			// Refresh active signal
			IF NOT _ServiceStates[nIndex].Alarm.Active THEN
				_ServiceStates[nIndex].Alarm.Active := TRUE;
				_ServiceStates[nIndex].Alarm.Acknowledged := FALSE;
				_ServiceStates[nIndex].Alarm.OccurrenceCount := _ServiceStates[nIndex].Alarm.OccurrenceCount + 1;
			END_IF
			M_ObserveServiceAlarm := TRUE;
			RETURN;
		END_IF

	// Update first empty slot index
	ELSIF nFirstEmpty = 0 THEN
		nFirstEmpty := nIndex;
	END_IF
END_FOR

IF nFirstEmpty = 0 THEN
	Overflow := TRUE;
	RETURN;
END_IF

M_LatchState(
	State := _ServiceStates[nFirstEmpty],
	Snapshot := Alarm,
	ServiceId := Alarm.ServiceId,
	DateTime := Alarm.DateTime);
_ServiceStates[nFirstEmpty].SeenThisCycle := TRUE;
M_ObserveServiceAlarm := TRUE;
END_METHOD

METHOD PUBLIC M_ProcessAcknowledgement
VAR_IN_OUT CONSTANT
	Request : ST_AlarmAckRequest;
END_VAR
VAR
	nIndex : UINT;
	bFound : BOOL;
END_VAR
_AckRequestOneShot(CLK := Request.bChangeRequest);

// Keep the response visible until the upper controller releases the request.
IF NOT Request.bChangeRequest THEN
	AckAccepted := FALSE;
	AckError := E_AlarmAckError.None;
	RETURN;
END_IF

IF NOT _AckRequestOneShot.Q THEN
	RETURN;
END_IF

AckResponseId := Request.RequestId;
AckAccepted := FALSE;
AckError := E_AlarmAckError.None;
bFound := FALSE;

IF Request.RequestId = 0 THEN
	AckError := E_AlarmAckError.InvalidRequestId;
	RETURN;
END_IF
IF Request.RequestId = _LastAckRequestId THEN
	AckError := E_AlarmAckError.DuplicateRequest;
	RETURN;
END_IF
_LastAckRequestId := Request.RequestId;

CASE Request.Command OF
	E_AlarmAckCommand.AcknowledgeOne:
		IF Request.MainErrorId = 0 THEN
			AckError := E_AlarmAckError.AlarmNotFound;
			RETURN;
		END_IF

		IF Request.ServiceId = 0 THEN
			FOR nIndex := 1 TO Param_Config.MaxConfiguredAlarmsPerModule DO
				IF _ConfiguredStates[nIndex].Latched
					AND (_ConfiguredStates[nIndex].Alarm.MainErrorId = Request.MainErrorId) THEN
					M_AcknowledgeState(State := _ConfiguredStates[nIndex]);
					bFound := TRUE;
					EXIT;
				END_IF
			END_FOR

			IF NOT bFound THEN
				FOR nIndex := 1 TO Param_Config.MaxHookAlarmsPerModule DO
					IF _HookStates[nIndex].Latched
						AND (_HookStates[nIndex].Alarm.MainErrorId = Request.MainErrorId) THEN
						M_AcknowledgeState(State := _HookStates[nIndex]);
						bFound := TRUE;
						EXIT;
					END_IF
				END_FOR
			END_IF
		ELSE
			FOR nIndex := 1 TO Param_Config.MaxServiceAlarmsPerModule DO
				IF _ServiceStates[nIndex].Latched
					AND (_ServiceStates[nIndex].Alarm.ServiceId = Request.ServiceId)
					AND (_ServiceStates[nIndex].Alarm.MainErrorId = Request.MainErrorId) THEN
					M_AcknowledgeState(State := _ServiceStates[nIndex]);
					bFound := TRUE;
					EXIT;
				END_IF
			END_FOR
		END_IF

		IF NOT bFound THEN
			AckError := E_AlarmAckError.AlarmNotFound;
			RETURN;
		END_IF

	E_AlarmAckCommand.AcknowledgeAll:
		FOR nIndex := 1 TO Param_Config.MaxConfiguredAlarmsPerModule DO
			IF _ConfiguredStates[nIndex].Latched THEN
				M_AcknowledgeState(State := _ConfiguredStates[nIndex]);
			END_IF
		END_FOR
		FOR nIndex := 1 TO Param_Config.MaxServiceAlarmsPerModule DO
			IF _ServiceStates[nIndex].Latched THEN
				M_AcknowledgeState(State := _ServiceStates[nIndex]);
			END_IF
		END_FOR

		FOR nIndex := 1 TO Param_Config.MaxHookAlarmsPerModule DO
			IF _HookStates[nIndex].Latched THEN
				M_AcknowledgeState(State := _HookStates[nIndex]);
			END_IF
		END_FOR
ELSE
	AckError := E_AlarmAckError.InvalidCommand;
	RETURN;
END_CASE

AckAccepted := TRUE;
END_METHOD

METHOD PUBLIC M_Publish
VAR_IN_OUT
	AlarmList : ARRAY[1..Param_Config.MaxPublishedModuleAlarms] OF ST_ExtAlarm;
END_VAR
VAR
	nIndex : UINT;
	nTarget : UINT;
END_VAR
MEMSET(ADR(AlarmList), 0, SIZEOF(AlarmList));
ConfiguredLatchedCount := 0;
ServiceLatchedCount := 0;
HookLatchedCount := 0;
nTarget := 1;

// Publish Service alarms first, configured alarms second, Hook alarms last.
FOR nIndex := 1 TO Param_Config.MaxServiceAlarmsPerModule DO
	IF NOT _ServiceStates[nIndex].Latched THEN
		CONTINUE;
	END_IF
	ServiceLatchedCount := ServiceLatchedCount + 1;
	IF nTarget > Param_Config.MaxPublishedModuleAlarms THEN
		Overflow := TRUE;
		CONTINUE;
	END_IF
	AlarmList[nTarget] := _ServiceStates[nIndex].Alarm;
	nTarget := nTarget + 1;
END_FOR

FOR nIndex := 1 TO Param_Config.MaxConfiguredAlarmsPerModule DO
	IF NOT _ConfiguredStates[nIndex].Latched THEN
		CONTINUE;
	END_IF
	ConfiguredLatchedCount := ConfiguredLatchedCount + 1;
	IF nTarget > Param_Config.MaxPublishedModuleAlarms THEN
		Overflow := TRUE;
		CONTINUE;
	END_IF
	AlarmList[nTarget] := _ConfiguredStates[nIndex].Alarm;
	nTarget := nTarget + 1;
END_FOR

FOR nIndex := 1 TO Param_Config.MaxHookAlarmsPerModule DO
	IF NOT _HookStates[nIndex].Latched THEN
		CONTINUE;
	END_IF
	HookLatchedCount := HookLatchedCount + 1;
	IF nTarget > Param_Config.MaxPublishedModuleAlarms THEN
		Overflow := TRUE;
		CONTINUE;
	END_IF
	AlarmList[nTarget] := _HookStates[nIndex].Alarm;
	nTarget := nTarget + 1;
END_FOR
END_METHOD

METHOD PRIVATE M_ResetAcknowledgement
AckResponseId := 0;
AckAccepted := FALSE;
AckError := E_AlarmAckError.None;
_LastAckRequestId := 0;
_AckRequestOneShot(CLK := FALSE);
END_METHOD

METHOD PUBLIC M_UpdateConfiguredAlarm
VAR_INPUT
	AlarmIndex : UINT;
	SampleValid : BOOL;
	ConditionMet : BOOL;
	UtcDateTime : STRING(20);
END_VAR
VAR_IN_OUT CONSTANT
	Alarm : ST_ExtAlarm;
END_VAR
IF (AlarmIndex < 1)
	OR (AlarmIndex > Param_Config.MaxConfiguredAlarmsPerModule)
	OR NOT SampleValid THEN
	RETURN;
END_IF

IF ConditionMet THEN
	IF NOT _ConfiguredStates[AlarmIndex].PreviousActive THEN
		IF NOT _ConfiguredStates[AlarmIndex].Latched THEN
			M_LatchState(
				State := _ConfiguredStates[AlarmIndex],
				Snapshot := Alarm,
				ServiceId := 0,
				DateTime := UtcDateTime);
		ELSE
			_ConfiguredStates[AlarmIndex].Alarm.Active := TRUE;
			_ConfiguredStates[AlarmIndex].Alarm.Acknowledged := FALSE;
			_ConfiguredStates[AlarmIndex].Alarm.OccurrenceCount := _ConfiguredStates[AlarmIndex].Alarm.OccurrenceCount + 1;
		END_IF
	END_IF
	_ConfiguredStates[AlarmIndex].Alarm.Active := TRUE;

ELSE
	IF _ConfiguredStates[AlarmIndex].PreviousActive
		AND _ConfiguredStates[AlarmIndex].Latched THEN
		_ConfiguredStates[AlarmIndex].Alarm.Active := FALSE;
		IF _ConfiguredStates[AlarmIndex].Alarm.Acknowledged THEN
			MEMSET(ADR(_ConfiguredStates[AlarmIndex]), 0, SIZEOF(_ConfiguredStates[AlarmIndex]));
		END_IF
	END_IF
END_IF

_ConfiguredStates[AlarmIndex].PreviousActive := ConditionMet;
END_METHOD

METHOD PUBLIC M_ObserveHookAlarm : BOOL
VAR_IN_OUT CONSTANT
	Alarm : ST_ExtAlarm;
END_VAR
VAR
	nIndex : UINT;
	nFirstEmpty : UINT;
END_VAR
M_ObserveHookAlarm := FALSE;
nFirstEmpty := 0;

IF (Alarm.ServiceId <> 0) OR (Alarm.MainErrorId = 0) THEN
	RETURN;
END_IF

FOR nIndex := 1 TO Param_Config.MaxHookAlarmsPerModule DO

	IF _HookStates[nIndex].Latched THEN

		IF (_HookStates[nIndex].Alarm.ServiceId = Alarm.ServiceId)
			AND (_HookStates[nIndex].Alarm.MainErrorId = Alarm.MainErrorId) THEN
			IF _HookStates[nIndex].SeenThisCycle THEN
				IF DuplicateId = 0 THEN
					DuplicateId := Alarm.MainErrorId;
				END_IF
				RETURN;
			END_IF
			_HookStates[nIndex].SeenThisCycle := TRUE;

			// A recurrence keeps the first snapshot and requires a fresh acknowledgement.
			IF NOT _HookStates[nIndex].Alarm.Active THEN
				_HookStates[nIndex].Alarm.Active := TRUE;
				_HookStates[nIndex].Alarm.Acknowledged := FALSE;
				_HookStates[nIndex].Alarm.OccurrenceCount := _HookStates[nIndex].Alarm.OccurrenceCount + 1;
			END_IF
			M_ObserveHookAlarm := TRUE;
			RETURN;
		END_IF

	// Reserve the first free slot without replacing a latched lifecycle.
	ELSIF nFirstEmpty = 0 THEN
		nFirstEmpty := nIndex;
	END_IF
END_FOR

IF nFirstEmpty = 0 THEN
	Overflow := TRUE;
	RETURN;
END_IF

M_LatchState(
	State := _HookStates[nFirstEmpty],
	Snapshot := Alarm,
	ServiceId := Alarm.ServiceId,
	DateTime := Alarm.DateTime);
_HookStates[nFirstEmpty].SeenThisCycle := TRUE;
M_ObserveHookAlarm := TRUE;
END_METHOD

METHOD PUBLIC M_SuppressHookAlarm
VAR_INPUT
	MainErrorId : UDINT;
END_VAR
VAR
	nIndex : UINT;
END_VAR
// Apply configuration ownership before acknowledgement, even when the source is invalid.
FOR nIndex := 1 TO Param_Config.MaxHookAlarmsPerModule DO
	IF _HookStates[nIndex].Latched AND (_HookStates[nIndex].Alarm.MainErrorId = MainErrorId) THEN
		MEMSET(ADR(_HookStates[nIndex]), 0, SIZEOF(_HookStates[nIndex]));
		RETURN;
	END_IF
END_FOR
END_METHOD

END_FUNCTION_BLOCK

// ---- POUs/10_Module/FB_ModuleBase.TcPOU
FUNCTION_BLOCK FB_ModuleBase EXTENDS FB_PackMLModeSet
VAR_INPUT
	ModuleCtrl : REFERENCE TO ST_ModuleCtrl;
	SystemContext : REFERENCE TO ST_SystemContext;
	HeartbeatIndex : UDINT;
	RuntimeConfig : REFERENCE TO ST_ModuleRuntimeConfig;
	VariableNodeReader : I_VariableNodeReader;
END_VAR

VAR_OUTPUT
	ModuleStatus : ST_ModuleStatus;
	ModuleVariableList : ARRAY[1..Param_Config.MaxModuleVariable] OF ST_ExtDescriptor;
	ModuleAlarmList : ARRAY[1..Param_Config.MaxPublishedModuleAlarms] OF ST_ExtAlarm;
	ModuleDataList : ARRAY[1..Param_Config.MaxModuleData] OF ST_ExtDescriptor;
END_VAR

VAR
	_CmdRequestOneShot : R_TRIG;
	_ModeRequestOneShot : R_TRIG;
	
	_ModuleId : UDINT;
	_ServiceContext : ST_ServiceContext;
	
	_HeartbeatTimer : TON;
	_LastHeartbeatIndex : UDINT;
	_IsControlSourceAlive : BOOL;
	_ConfiguredSnapshot : FB_ConfigValueSnapshotReader;
	_AlarmManager : FB_ModuleAlarmManager;
	_InAlarmHook : BOOL;
	_InVariableHook : BOOL;
	_ConfiguredVariableCount : UINT;
	_ServiceCoordinator : FB_ServiceCoordinator;
	_ServiceRegistrationAttempted : BOOL;
END_VAR

METHOD PROTECTED FINAL H_OnAborting : E_PackMLHookResult
VAR_INPUT
	bFirstScan : BOOL;
END_VAR
H_OnAborting := E_PackMLHookResult.Busy;
IF _ServiceCoordinator.AllAborted THEN
	H_OnAborting := E_PackMLHookResult.Done;
END_IF
END_METHOD

METHOD PROTECTED FINAL H_OnClearing : E_PackMLHookResult
VAR_INPUT
	bFirstScan : BOOL;
END_VAR
H_OnClearing := E_PackMLHookResult.Busy;
IF _ServiceCoordinator.AllStopped THEN
	H_OnClearing := E_PackMLHookResult.Done;
END_IF
END_METHOD

METHOD PROTECTED FINAL H_OnIdle
VAR_INPUT
	bFirstScan	: BOOL;
END_VAR
// Transfer to execute automatically
RequestCommand(E_PackMLCommand.Start);
END_METHOD

METHOD PROTECTED FINAL H_OnResetting : E_PackMLHookResult
VAR_INPUT
	bFirstScan : BOOL;
END_VAR
H_OnResetting := E_PackMLHookResult.Busy;
IF _ServiceCoordinator.AllIdle THEN
	H_OnResetting := E_PackMLHookResult.Done;
END_IF
END_METHOD

METHOD PROTECTED FINAL H_OnStopping : E_PackMLHookResult
VAR_INPUT
	bFirstScan : BOOL;
END_VAR
H_OnStopping := E_PackMLHookResult.Busy;
IF _ServiceCoordinator.AllStopped THEN
	H_OnStopping := E_PackMLHookResult.Done;
END_IF
END_METHOD

METHOD PROTECTED H_RegisterServices
// Derived Modules register persistent Service storage once.
END_METHOD

METHOD PROTECTED H_UpdateAlarm
// Optional Module extension; submitted values belong to this scan.
END_METHOD

METHOD PROTECTED H_UpdateBaseUnit
VAR_INPUT
END_VAR
END_METHOD

METHOD PROTECTED H_UpdateService
VAR_INPUT
END_VAR
END_METHOD

METHOD PROTECTED H_UpdateVariable
// Optional Module extension; submitted values belong to this scan.
END_METHOD

METHOD PROTECTED FINAL M_AddAlarm : BOOL
VAR_INPUT
	MainErrorId : UDINT;
	SourceErrorId : UDINT;
	Message : STRING;
	Path : STRING(255);
	Severity : E_Severity;
END_VAR
VAR
	nIndex : UINT;
	Alarm : ST_ExtAlarm;
END_VAR
M_AddAlarm := FALSE;
IF NOT _InAlarmHook OR (MainErrorId = 0) THEN
	RETURN;
END_IF
IF __ISVALIDREF(RuntimeConfig) THEN
	IF RuntimeConfig.Valid THEN
		FOR nIndex := 1 TO RuntimeConfig.AlarmCount DO
			IF RuntimeConfig.AlarmBindings[nIndex].Definition.MainErrorId = MainErrorId THEN
				M_AddAlarm := TRUE; // JSON owns the complete definition, even without a valid sample.
				RETURN;
			END_IF
		END_FOR
	END_IF
END_IF
MEMSET(ADR(Alarm), 0, SIZEOF(Alarm));
Alarm.MainErrorId := MainErrorId;
Alarm.SourceErrorId := SourceErrorId;
Alarm.Message := Message;
Alarm.Path := Path;
Alarm.Severity := Severity;
Alarm.DateTime := _ServiceContext.UtcDateTime;
M_AddAlarm := _AlarmManager.M_ObserveHookAlarm(Alarm := Alarm);
END_METHOD

METHOD PROTECTED FINAL M_AddVariable : BOOL
VAR_INPUT
	Id : UDINT;
	Name : STRING(30);
	DataType : E_DescriptorType;
	Unit : STRING(10);
	Value : STRING(80);
END_VAR
VAR
	nIndex : UINT;
END_VAR
M_AddVariable := FALSE;
IF NOT _InVariableHook OR (Id = 0) THEN
	RETURN;
END_IF
FOR nIndex := 1 TO ModuleStatus.Variable.PublishedCount DO
	IF ModuleVariableList[nIndex].Id = Id THEN
		IF nIndex <= _ConfiguredVariableCount THEN
			M_AddVariable := TRUE; // JSON ownership is not a duplicate submission.
		ELSIF ModuleStatus.Variable.DuplicateId = 0 THEN
			ModuleStatus.Variable.DuplicateId := Id;
		END_IF
		RETURN;
	END_IF
END_FOR
IF ModuleStatus.Variable.PublishedCount >= Param_Config.MaxModuleVariable THEN
	ModuleStatus.Variable.Overflow := TRUE;
	RETURN;
END_IF
ModuleStatus.Variable.PublishedCount := ModuleStatus.Variable.PublishedCount + 1;
nIndex := ModuleStatus.Variable.PublishedCount;
ModuleVariableList[nIndex].Id := Id;
ModuleVariableList[nIndex].Name := Name;
ModuleVariableList[nIndex].DataType := DataType;
ModuleVariableList[nIndex].Unit := Unit;
ModuleVariableList[nIndex].Value := Value;
M_AddVariable := TRUE;
END_METHOD

METHOD PRIVATE M_CheckHeartbeat
VAR_INPUT
END_VAR

VAR
	bLooseHeartbeat : BOOL;
	HeartbeatTimeout : TIME;
END_VAR
HeartbeatTimeout := SystemContext.ModuleHeartbeatTimeout;
IF HeartbeatTimeout <= T#0S THEN
	HeartbeatTimeout := Param_Config.ModuleHeartbeat_Timeout;
END_IF

// Heartbeats check
bLooseHeartbeat := _LastHeartbeatIndex = HeartbeatIndex;
IF bLooseHeartbeat THEN
	_HeartbeatTimer(IN := TRUE, PT := HeartbeatTimeout);
ELSE
	_HeartbeatTimer(IN := FALSE, PT := HeartbeatTimeout);
END_IF

// Update Last Heartbeat Index
_LastHeartbeatIndex := HeartbeatIndex;

// Update Is ControlSource Alive status
_IsControlSourceAlive := NOT _HeartbeatTimer.Q;
END_METHOD

METHOD PRIVATE M_PublishAlarmState
_AlarmManager.M_Publish(AlarmList := ModuleAlarmList);
ModuleStatus.Alarm.AckResponseId := _AlarmManager.AckResponseId;
ModuleStatus.Alarm.AckAccepted := _AlarmManager.AckAccepted;
ModuleStatus.Alarm.AckError := _AlarmManager.AckError;
ModuleStatus.Alarm.ConfiguredLatchedCount := _AlarmManager.ConfiguredLatchedCount;
ModuleStatus.Alarm.Overflow := _AlarmManager.Overflow;
ModuleStatus.Alarm.ServiceLatchedCount := _AlarmManager.ServiceLatchedCount;
ModuleStatus.Alarm.HookLatchedCount := _AlarmManager.HookLatchedCount;
ModuleStatus.Alarm.DuplicateId := _AlarmManager.DuplicateId;
END_METHOD

METHOD PROTECTED FINAL M_RegisterService : BOOL
VAR_INPUT
	ServiceId : UDINT;
	AllowCompositeCall : BOOL;
	UpperParam : ANY;
	EffectiveParam : ANY;
END_VAR
VAR_IN_OUT
	UpperCtrl : ST_ServiceCtrl;
	EffectiveCtrl : ST_ServiceCtrl;
	Status : ST_ServiceStatus;
END_VAR
M_RegisterService := _ServiceCoordinator.M_Register(
	ServiceId := ServiceId,
	AllowCompositeCall := AllowCompositeCall,
	UpperCtrl := UpperCtrl,
	EffectiveCtrl := EffectiveCtrl,
	UpperParam := UpperParam,
	EffectiveParam := EffectiveParam,
	Status := Status);
END_METHOD

METHOD PRIVATE M_UpdateAlarmState
VAR
	nAlarm : UINT;
	nSource : UINT;
	nRevision : UDINT;
	fValue : LREAL;
	bValid : BOOL;
	bConditionMet : BOOL;
	Alarm : ST_ExtAlarm;
END_VAR
nRevision := 0;
IF __ISVALIDREF(RuntimeConfig) THEN
	IF RuntimeConfig.Valid THEN
		nRevision := RuntimeConfig.Revision;
	END_IF
END_IF
_AlarmManager.M_BeginCycle(
	ModuleId := _ModuleId,
	ConfigurationRevision := nRevision);

// Remove identities now owned by JSON before an acknowledgement can find a stale Hook event.
IF __ISVALIDREF(RuntimeConfig) THEN
	IF RuntimeConfig.Valid THEN
		FOR nAlarm := 1 TO RuntimeConfig.AlarmCount DO
			_AlarmManager.M_SuppressHookAlarm(
				MainErrorId := RuntimeConfig.AlarmBindings[nAlarm].Definition.MainErrorId);
		END_FOR
	END_IF
END_IF

// Process acknowledgements before evaluating this cycle so AckAll cannot consume
// a new event that the upper controller has not observed yet.
_AlarmManager.M_ProcessAcknowledgement(Request := ModuleCtrl.AlarmAckRequest);

IF __ISVALIDREF(RuntimeConfig) THEN
	IF RuntimeConfig.Valid AND _ConfiguredSnapshot.Ready THEN
		FOR nAlarm := 1 TO RuntimeConfig.AlarmCount DO
			nSource := RuntimeConfig.VariableCount + nAlarm;
			fValue := _ConfiguredSnapshot.M_GetLReal(SourceIndex := nSource, Valid => bValid);
			bConditionMet := FALSE;
			IF bValid THEN
				bConditionMet := F_AlarmConditionMet(
					Value := fValue,
					Operator := RuntimeConfig.AlarmBindings[nAlarm].Definition.Operator,
					Threshold := RuntimeConfig.AlarmBindings[nAlarm].Definition.Threshold,
					Tolerance := RuntimeConfig.AlarmBindings[nAlarm].Definition.Tolerance);
			END_IF

			MEMSET(ADR(Alarm), 0, SIZEOF(Alarm));
			Alarm.ModuleId := _ModuleId;
			Alarm.ServiceId := 0;
			Alarm.MainErrorId := RuntimeConfig.AlarmBindings[nAlarm].Definition.MainErrorId;
			Alarm.SourceErrorId := RuntimeConfig.AlarmBindings[nAlarm].Definition.SourceErrorId;
			Alarm.Message := RuntimeConfig.AlarmBindings[nAlarm].Definition.Message;
			Alarm.Path := RuntimeConfig.AlarmBindings[nAlarm].Definition.Source;
			Alarm.Severity := RuntimeConfig.AlarmBindings[nAlarm].Definition.Severity;
			_AlarmManager.M_UpdateConfiguredAlarm(
				AlarmIndex := nAlarm,
				SampleValid := bValid,
				ConditionMet := bConditionMet,
				Alarm := Alarm,
				UtcDateTime := _ServiceContext.UtcDateTime);
		END_FOR
	END_IF
END_IF

_InAlarmHook := TRUE;
H_UpdateAlarm();
_InAlarmHook := FALSE;

M_UpdateServiceAlarms();
_AlarmManager.M_EndCycle();
END_METHOD

METHOD PRIVATE M_UpdateConfiguredVariableList
VAR
	nVariable : UINT;
	bValid : BOOL;
END_VAR
IF NOT __ISVALIDREF(RuntimeConfig) THEN
	RETURN;
END_IF
IF NOT RuntimeConfig.Valid THEN
	RETURN;
END_IF

FOR nVariable := 1 TO RuntimeConfig.VariableCount DO
	ModuleVariableList[nVariable].Id := RuntimeConfig.VariableBindings[nVariable].Definition.Id;
	ModuleVariableList[nVariable].Name := RuntimeConfig.VariableBindings[nVariable].Definition.Name;
	ModuleVariableList[nVariable].DataType := F_ConfigDataTypeToDescriptor(
		DataType := RuntimeConfig.VariableBindings[nVariable].Definition.DataType);
	ModuleVariableList[nVariable].Unit := RuntimeConfig.VariableBindings[nVariable].Definition.Unit;
	ModuleVariableList[nVariable].Value := _ConfiguredSnapshot.M_GetValueString(
		SourceIndex := nVariable,
		Valid => bValid);
END_FOR
_ConfiguredVariableCount := RuntimeConfig.VariableCount;
ModuleStatus.Variable.PublishedCount := _ConfiguredVariableCount;
END_METHOD

METHOD PROTECTED FINAL M_UpdateModule
IF NOT _ServiceRegistrationAttempted THEN
	_ServiceRegistrationAttempted := TRUE;
	_ServiceCoordinator.M_BeginRegistration();
	H_RegisterServices();
	_ServiceCoordinator.M_Seal();
END_IF

M_CheckHeartbeat();
ModuleStatus.IsControlSourceAlive := _IsControlSourceAlive;

// Update module state machine
PackMLIn := ModuleCtrl.PackMLIn;
SUPER^();

IF __ISVALIDREF(RuntimeConfig) THEN
	_ModuleId := RuntimeConfig.ModuleId;
	_ConfiguredSnapshot(
		RuntimeConfig := RuntimeConfig,
		VariableNodeReader := VariableNodeReader);
	ModuleStatus.ModuleId := _ModuleId;
	ModuleStatus.Enabled := RuntimeConfig.Enabled;
	ModuleStatus.ModuleType := RuntimeConfig.ModuleType;
END_IF

_ServiceContext.ModuleId := _ModuleId;
_ServiceContext.UtcDateTime := SystemContext.UtcDateTime;

// Update service state machine
_ServiceCoordinator.M_PrepareCycle(
	ModuleInExecute := PackMLOut.eStateCurrent = E_PackMLState.Execute,
	ModuleCtrl := ModuleCtrl);
H_UpdateService();

// Update base unit state machine
H_UpdateBaseUnit();

// Capture the status set produced by this scan for framework aggregation and
// for the Module PackML transition checks in the next scan.
_ServiceCoordinator.M_ObserveCycle();

_CmdRequestOneShot(CLK:= PackMLIn.bCommandChangeRequest, Q=> );
_ModeRequestOneShot(CLK:= PackMLIn.bModeChangeRequest, Q=> );

// Updata status
IF _CmdRequestOneShot.Q OR _ModeRequestOneShot.Q THEN
	ModuleStatus.ResponseId := ModuleCtrl.RequestId;
END_IF
ModuleStatus.PackMLOut := PackMLOut;

M_UpdateAlarmState();
M_PublishAlarmState();
M_UpdateServiceDataList();
M_UpdateVariableList();
END_METHOD

METHOD PRIVATE M_UpdateServiceAlarms
VAR
	nServiceIndex : UINT;
	nErrorIndex : UINT;
	ServiceStatus : ST_ServiceStatus;
END_VAR
// Submit currently observable Service errors. The manager owns lifecycle state
// and marks identities not observed in this scan inactive during M_EndCycle.
FOR nServiceIndex := 1 TO _ServiceCoordinator.RegisteredCount DO
	IF NOT _ServiceCoordinator.M_GetServiceStatusByIndex(
		Index := nServiceIndex,
		Status => ServiceStatus) THEN
		CONTINUE;
	END_IF
	FOR nErrorIndex := 1 TO Param_Config.MaxServiceError DO
		IF ServiceStatus.ErrorList[nErrorIndex].MainErrorId <> 0 THEN
			_AlarmManager.M_ObserveServiceAlarm(
				Alarm := ServiceStatus.ErrorList[nErrorIndex]);
		END_IF
	END_FOR
END_FOR
END_METHOD

METHOD PRIVATE M_UpdateServiceDataList
VAR
	nServiceIndex : UINT;
	nDataIndex : UINT;
	nPublishedIndex : UINT;
	bDuplicate : BOOL;
	DataId : UDINT;
	ServiceStatus : ST_ServiceStatus;
END_VAR
MEMSET(ADR(ModuleDataList), 0, SIZEOF(ModuleDataList));
MEMSET(ADR(ModuleStatus.Data), 0, SIZEOF(ModuleStatus.Data));

FOR nServiceIndex := 1 TO _ServiceCoordinator.RegisteredCount DO
	IF NOT _ServiceCoordinator.M_GetServiceStatusByIndex(
		Index := nServiceIndex,
		Status => ServiceStatus) THEN
		CONTINUE;
	END_IF
	IF ServiceStatus.Data.Overflow THEN
		ModuleStatus.Data.Overflow := TRUE;
	END_IF

	FOR nDataIndex := 1 TO Param_Config.MaxServiceData DO
		DataId := ServiceStatus.Data.DataList[nDataIndex].Id;
		IF DataId = 0 THEN
			CONTINUE;
		END_IF

		bDuplicate := FALSE;
		FOR nPublishedIndex := 1 TO ModuleStatus.Data.PublishedCount DO
			IF ModuleDataList[nPublishedIndex].Id = DataId THEN
				bDuplicate := TRUE;
				EXIT;
			END_IF
		END_FOR

		IF bDuplicate THEN
			IF ModuleStatus.Data.DuplicateId = 0 THEN
				ModuleStatus.Data.DuplicateId := DataId;
			END_IF
			CONTINUE;
		END_IF

		IF ModuleStatus.Data.PublishedCount >= Param_Config.MaxModuleData THEN
			ModuleStatus.Data.Overflow := TRUE;
			CONTINUE;
		END_IF

		ModuleStatus.Data.PublishedCount := ModuleStatus.Data.PublishedCount + 1;
		ModuleDataList[ModuleStatus.Data.PublishedCount] :=
			ServiceStatus.Data.DataList[nDataIndex];
	END_FOR
END_FOR
END_METHOD

METHOD PRIVATE M_UpdateVariableList
MEMSET(ADR(ModuleVariableList), 0, SIZEOF(ModuleVariableList));
MEMSET(ADR(ModuleStatus.Variable), 0, SIZEOF(ModuleStatus.Variable));
_ConfiguredVariableCount := 0;
M_UpdateConfiguredVariableList();
_InVariableHook := TRUE;
H_UpdateVariable();
_InVariableHook := FALSE;
END_METHOD

END_FUNCTION_BLOCK

// ---- POUs/10_Module/FB_ServiceCoordinator.TcPOU
FUNCTION_BLOCK FB_ServiceCoordinator
VAR
	_Entries : ARRAY[1..Param_Config.MaxServicesPerModule] OF ST_ServiceRegistrationEntry;
	_RegisteredCount : UINT;
	_RegistrationStarted : BOOL;
	_Sealed : BOOL;
	_RegistrationError : E_ServiceRegistrationError;
	_FailedServiceId : UDINT;
	_AllIdle : BOOL;
	_AllStopped : BOOL;
	_AllAborted : BOOL;
	_JsonDataType : FB_JsonReadWriteDataType;
END_VAR

PROPERTY PUBLIC FINAL AllAborted : BOOL
GET
AllAborted := _AllAborted;
END_GET
END_PROPERTY

PROPERTY PUBLIC FINAL AllIdle : BOOL
GET
AllIdle := _AllIdle;
END_GET
END_PROPERTY

PROPERTY PUBLIC FINAL AllStopped : BOOL
GET
AllStopped := _AllStopped;
END_GET
END_PROPERTY

PROPERTY PUBLIC FINAL FailedServiceId : UDINT
GET
FailedServiceId := _FailedServiceId;
END_GET
END_PROPERTY

METHOD PUBLIC FINAL M_BeginRegistration : BOOL
M_BeginRegistration := FALSE;
IF _RegistrationStarted THEN
	M_SetRegistrationError(Error := E_ServiceRegistrationError.RegistrationAlreadyStarted, ServiceId := 0);
	RETURN;
END_IF
MEMSET(ADR(_Entries), 0, SIZEOF(_Entries));
_RegisteredCount := 0;
_Sealed := FALSE;
_RegistrationError := E_ServiceRegistrationError.None;
_FailedServiceId := 0;
_AllIdle := FALSE;
_AllStopped := FALSE;
_AllAborted := FALSE;
_RegistrationStarted := TRUE;
M_BeginRegistration := TRUE;
END_METHOD

METHOD PRIVATE M_FindIndexByServiceId : UINT
VAR_INPUT
	ServiceId : UDINT;
END_VAR
VAR
	nIndex : UINT;
END_VAR
M_FindIndexByServiceId := 0;
IF ServiceId = 0 THEN RETURN; END_IF
FOR nIndex := 1 TO _RegisteredCount DO
	IF _Entries[nIndex].InUse AND (_Entries[nIndex].ServiceId = ServiceId) THEN
		M_FindIndexByServiceId := nIndex;
		RETURN;
	END_IF
END_FOR
END_METHOD

METHOD PUBLIC FINAL M_GetCompositeOwnershipState : E_CompositeOwnershipState
VAR_INPUT
	CompositeServiceId : UDINT;
END_VAR
VAR
	nIndex : UINT;
END_VAR
M_GetCompositeOwnershipState := E_CompositeOwnershipState.None;
nIndex := M_FindIndexByServiceId(ServiceId := CompositeServiceId);
IF (nIndex = 0) OR NOT _Entries[nIndex].IsComposite THEN RETURN; END_IF
M_GetCompositeOwnershipState := _Entries[nIndex].OwnershipState;
END_METHOD

METHOD PUBLIC FINAL M_GetInternalCommandState : E_ServiceInternalCommandState
VAR_INPUT
	CallerServiceId : UDINT;
	TargetServiceId : UDINT;
END_VAR
VAR
	nCallerIndex : UINT;
	nTargetIndex : UINT;
END_VAR
M_GetInternalCommandState := E_ServiceInternalCommandState.None;
nCallerIndex := M_FindIndexByServiceId(ServiceId := CallerServiceId);
nTargetIndex := M_FindIndexByServiceId(ServiceId := TargetServiceId);
IF (nCallerIndex = 0) OR (nTargetIndex = 0) THEN RETURN; END_IF
IF NOT M_IsDeclaredDependency(CompositeIndex := nCallerIndex, TargetServiceId := TargetServiceId) THEN RETURN; END_IF
IF (_Entries[nTargetIndex].CompositeOwnerServiceId <> CallerServiceId)
	AND (_Entries[nTargetIndex].InternalCommandState <> E_ServiceInternalCommandState.Cancelled) THEN RETURN; END_IF
M_GetInternalCommandState := _Entries[nTargetIndex].InternalCommandState;
END_METHOD

METHOD PUBLIC FINAL M_GetServiceSnapshotById : BOOL
VAR_INPUT
	ServiceId : UDINT;
END_VAR
VAR_OUTPUT
	Snapshot : ST_ServiceExecutionSnapshot;
END_VAR
VAR
	nIndex : UINT;
END_VAR
M_GetServiceSnapshotById := FALSE;
MEMSET(ADR(Snapshot), 0, SIZEOF(Snapshot));
nIndex := M_FindIndexByServiceId(ServiceId := ServiceId);
IF nIndex = 0 THEN RETURN; END_IF
Snapshot := _Entries[nIndex].ObservedSnapshot;
M_GetServiceSnapshotById := Snapshot.Valid;
END_METHOD

METHOD PUBLIC FINAL M_GetServiceStatusByIndex : BOOL
VAR_INPUT
	Index : UINT;
END_VAR
VAR_OUTPUT
	Status : ST_ServiceStatus;
END_VAR
VAR
	pStatus : POINTER TO ST_ServiceStatus;
END_VAR
M_GetServiceStatusByIndex := FALSE;
MEMSET(ADR(Status), 0, SIZEOF(Status));
IF (Index = 0) OR (Index > _RegisteredCount) THEN RETURN; END_IF
IF NOT _Entries[Index].InUse OR (_Entries[Index].StatusAddress = 0) THEN RETURN; END_IF
pStatus := _Entries[Index].StatusAddress;
Status := pStatus^;
M_GetServiceStatusByIndex := TRUE;
END_METHOD

METHOD PRIVATE M_IsDeclaredDependency : BOOL
VAR_INPUT
	CompositeIndex : UINT;
	TargetServiceId : UDINT;
END_VAR
VAR
	nDependency : UINT;
	pDependencies : POINTER TO UDINT;
END_VAR
M_IsDeclaredDependency := FALSE;
IF (CompositeIndex = 0) OR (CompositeIndex > _RegisteredCount)
	OR NOT _Entries[CompositeIndex].IsComposite
	OR (_Entries[CompositeIndex].CompositeDependenciesAddress = 0) THEN RETURN; END_IF

pDependencies := _Entries[CompositeIndex].CompositeDependenciesAddress;
FOR nDependency := 1 TO _Entries[CompositeIndex].CompositeDependencyCount DO
	IF pDependencies[nDependency - 1] = TargetServiceId THEN
		M_IsDeclaredDependency := TRUE;
		RETURN;
	END_IF
END_FOR
END_METHOD

METHOD PUBLIC FINAL M_ObserveCycle
VAR
	nIndex : UINT;
	pStatus : POINTER TO ST_ServiceStatus;
END_VAR
_AllIdle := FALSE;
_AllStopped := FALSE;
_AllAborted := FALSE;
IF NOT Ready OR (_RegisteredCount = 0) THEN RETURN; END_IF
_AllIdle := TRUE;
_AllStopped := TRUE;
_AllAborted := TRUE;
FOR nIndex := 1 TO _RegisteredCount DO
	pStatus := _Entries[nIndex].StatusAddress;
	_Entries[nIndex].ObservedSnapshot.Valid := TRUE;
	_Entries[nIndex].ObservedSnapshot.ServiceId := _Entries[nIndex].ServiceId;
	_Entries[nIndex].ObservedSnapshot.ResponseId := pStatus^.ResponseId;
	_Entries[nIndex].ObservedSnapshot.PackMLOut := pStatus^.PackMLOut;
	_Entries[nIndex].ObservedSnapshot.ExecuteSubState := pStatus^.ExecuteSubState;
	_Entries[nIndex].ObservedSnapshot.CompletionBehavior := pStatus^.CompletionBehavior;
	IF (_Entries[nIndex].InternalCommandState = E_ServiceInternalCommandState.RequestHigh)
		AND (pStatus^.ResponseId = _Entries[nIndex].InternalRequestId) THEN
		IF pStatus^.PackMLOut.bCommandAccepted THEN
			_Entries[nIndex].InternalCommandState := E_ServiceInternalCommandState.Accepted;
			_Entries[nIndex].InternalRequestMustGoLow := TRUE;
		ELSIF pStatus^.PackMLOut.bCommandRejected THEN
			_Entries[nIndex].InternalCommandState := E_ServiceInternalCommandState.Rejected;
			_Entries[nIndex].InternalRequestMustGoLow := TRUE;
		END_IF
	END_IF
	_AllIdle := _AllIdle AND (pStatus^.PackMLOut.eStateCurrent = E_PackMLState.Idle);
	_AllStopped := _AllStopped AND (pStatus^.PackMLOut.eStateCurrent = E_PackMLState.Stopped);
	_AllAborted := _AllAborted AND (pStatus^.PackMLOut.eStateCurrent = E_PackMLState.Aborted);
END_FOR
END_METHOD

METHOD PUBLIC FINAL M_PrepareCycle
VAR_INPUT
	ModuleInExecute : BOOL;
	ModuleCtrl : REFERENCE TO ST_ModuleCtrl;
END_VAR
VAR
	nIndex : UINT;
	pUpperCtrl : POINTER TO ST_ServiceCtrl;
	pEffectiveCtrl : POINTER TO ST_ServiceCtrl;
	bUpperCommandHigh : BOOL;
	bUpperModeHigh : BOOL;
	bNewStartRequest : BOOL;
END_VAR
IF Ready AND ModuleInExecute THEN
	M_ProcessOwnershipRequests();
ELSIF Ready THEN
	FOR nIndex := 1 TO _RegisteredCount DO
		IF _Entries[nIndex].OwnershipState = E_CompositeOwnershipState.Pending THEN
			_Entries[nIndex].OwnershipState := E_CompositeOwnershipState.Cancelled;
		END_IF
	END_FOR
END_IF
FOR nIndex := 1 TO _RegisteredCount DO
	pUpperCtrl := _Entries[nIndex].UpperCtrlAddress;
	pEffectiveCtrl := _Entries[nIndex].EffectiveCtrlAddress;
	IF NOT Ready THEN
		pEffectiveCtrl^.PackMLIn.bCommandChangeRequest := FALSE;
		pEffectiveCtrl^.PackMLIn.bModeChangeRequest := FALSE;
		CONTINUE;
	END_IF
	bUpperCommandHigh := pUpperCtrl^.PackMLIn.bCommandChangeRequest;
	bUpperModeHigh := pUpperCtrl^.PackMLIn.bModeChangeRequest;
	IF NOT ModuleInExecute THEN
		IF (_Entries[nIndex].InternalCommandState = E_ServiceInternalCommandState.Queued)
			OR (_Entries[nIndex].InternalCommandState = E_ServiceInternalCommandState.RequestHigh)
			OR _Entries[nIndex].InternalRequestMustGoLow THEN
			_Entries[nIndex].InternalCommandState := E_ServiceInternalCommandState.Cancelled;
			_Entries[nIndex].InternalRequestMustGoLow := FALSE;
		END_IF
		pEffectiveCtrl^.RequestId := ModuleCtrl.RequestId;
		pEffectiveCtrl^.PackMLIn := ModuleCtrl.PackMLIn;
		IF bUpperCommandHigh THEN _Entries[nIndex].UpperCommandBlockedUntilFalse := TRUE; END_IF
		IF bUpperModeHigh THEN _Entries[nIndex].UpperModeBlockedUntilFalse := TRUE; END_IF
		_Entries[nIndex].UpperCommandWasHigh := bUpperCommandHigh;
		_Entries[nIndex].UpperModeWasHigh := bUpperModeHigh;
		CONTINUE;
	END_IF
	IF NOT bUpperCommandHigh THEN _Entries[nIndex].UpperCommandBlockedUntilFalse := FALSE; END_IF
	IF NOT bUpperModeHigh THEN _Entries[nIndex].UpperModeBlockedUntilFalse := FALSE; END_IF
	IF _Entries[nIndex].CompositeOwnerServiceId <> 0 THEN
		IF bUpperCommandHigh THEN _Entries[nIndex].UpperCommandBlockedUntilFalse := TRUE; END_IF
		IF bUpperModeHigh THEN _Entries[nIndex].UpperModeBlockedUntilFalse := TRUE; END_IF
		pEffectiveCtrl^.PackMLIn.eMode := E_PackMLMode.Unknown;
		pEffectiveCtrl^.PackMLIn.bModeChangeRequest := FALSE;
		IF _Entries[nIndex].InternalRequestMustGoLow THEN
			pEffectiveCtrl^.PackMLIn.eCommand := E_PackMLCommand.None;
			pEffectiveCtrl^.PackMLIn.bCommandChangeRequest := FALSE;
			_Entries[nIndex].InternalRequestMustGoLow := FALSE;
		ELSIF _Entries[nIndex].InternalCommandState = E_ServiceInternalCommandState.Queued THEN
			pEffectiveCtrl^.RequestId := _Entries[nIndex].InternalRequestId;
			pEffectiveCtrl^.PackMLIn.eCommand := _Entries[nIndex].InternalCommand;
			pEffectiveCtrl^.PackMLIn.bCommandChangeRequest := TRUE;
			_Entries[nIndex].InternalCommandState := E_ServiceInternalCommandState.RequestHigh;
		ELSIF _Entries[nIndex].InternalCommandState = E_ServiceInternalCommandState.RequestHigh THEN
			pEffectiveCtrl^.RequestId := _Entries[nIndex].InternalRequestId;
			pEffectiveCtrl^.PackMLIn.eCommand := _Entries[nIndex].InternalCommand;
			pEffectiveCtrl^.PackMLIn.bCommandChangeRequest := TRUE;
		ELSE
			pEffectiveCtrl^.PackMLIn.eCommand := E_PackMLCommand.None;
			pEffectiveCtrl^.PackMLIn.bCommandChangeRequest := FALSE;
		END_IF
		_Entries[nIndex].UpperCommandWasHigh := bUpperCommandHigh;
		_Entries[nIndex].UpperModeWasHigh := bUpperModeHigh;
		CONTINUE;
	END_IF
	pEffectiveCtrl^ := pUpperCtrl^;
	IF _Entries[nIndex].UpperCommandBlockedUntilFalse THEN
		pEffectiveCtrl^.PackMLIn.bCommandChangeRequest := FALSE;
	ELSE
		bNewStartRequest := bUpperCommandHigh AND NOT _Entries[nIndex].UpperCommandWasHigh
			AND (pUpperCtrl^.PackMLIn.eCommand = E_PackMLCommand.Start);
		IF bNewStartRequest THEN
			MEMCPY(destAddr := _Entries[nIndex].EffectiveParamAddress,
				srcAddr := _Entries[nIndex].UpperParamAddress, n := _Entries[nIndex].ParameterSize);
		END_IF
	END_IF
	IF _Entries[nIndex].UpperModeBlockedUntilFalse THEN
		pEffectiveCtrl^.PackMLIn.bModeChangeRequest := FALSE;
	END_IF
	_Entries[nIndex].UpperCommandWasHigh := bUpperCommandHigh;
	_Entries[nIndex].UpperModeWasHigh := bUpperModeHigh;
END_FOR
END_METHOD

METHOD PRIVATE M_ProcessOwnershipRequests
VAR
	nOrder : UINT;
	nIndex : UINT;
	nCandidateIndex : UINT;
	nDependency : UINT;
	nDependencyIndex : UINT;
	nLastServiceId : UDINT;
	nCandidateServiceId : UDINT;
	pDependencies : POINTER TO UDINT;
	bConflict : BOOL;
	bNotIdle : BOOL;
	bUnsupported : BOOL;
END_VAR
nLastServiceId := 0;
FOR nOrder := 1 TO _RegisteredCount DO
	nCandidateIndex := 0;
	nCandidateServiceId := 0;
	FOR nIndex := 1 TO _RegisteredCount DO
		IF (_Entries[nIndex].OwnershipState = E_CompositeOwnershipState.Pending)
			AND (_Entries[nIndex].ServiceId > nLastServiceId)
			AND ((nCandidateIndex = 0) OR (_Entries[nIndex].ServiceId < nCandidateServiceId)) THEN
			nCandidateIndex := nIndex;
			nCandidateServiceId := _Entries[nIndex].ServiceId;
		END_IF
	END_FOR
	IF nCandidateIndex = 0 THEN EXIT; END_IF
	nLastServiceId := nCandidateServiceId;
	bConflict := FALSE;
	bNotIdle := FALSE;
	bUnsupported := FALSE;
	pDependencies := _Entries[nCandidateIndex].CompositeDependenciesAddress;
	FOR nDependency := 1 TO _Entries[nCandidateIndex].CompositeDependencyCount DO
		nDependencyIndex := M_FindIndexByServiceId(ServiceId := pDependencies[nDependency - 1]);
		IF _Entries[nDependencyIndex].CompositeOwnerServiceId <> 0 THEN
			bConflict := TRUE;
		ELSIF NOT _Entries[nDependencyIndex].ObservedSnapshot.Valid
			OR (_Entries[nDependencyIndex].ObservedSnapshot.PackMLOut.eStateCurrent <> E_PackMLState.Idle) THEN
			bNotIdle := TRUE;
		ELSIF _Entries[nDependencyIndex].ObservedSnapshot.CompletionBehavior
			<> E_ServiceCompletionBehavior.NaturalCompletion THEN
			bUnsupported := TRUE;
		END_IF
	END_FOR
	IF bConflict THEN
		_Entries[nCandidateIndex].OwnershipState := E_CompositeOwnershipState.RejectedConflict;
	ELSIF bUnsupported THEN
		_Entries[nCandidateIndex].OwnershipState := E_CompositeOwnershipState.RejectedUnsupportedCompletionBehavior;
	ELSIF bNotIdle THEN
		_Entries[nCandidateIndex].OwnershipState := E_CompositeOwnershipState.RejectedDependencyNotIdle;
	ELSE
		FOR nDependency := 1 TO _Entries[nCandidateIndex].CompositeDependencyCount DO
			nDependencyIndex := M_FindIndexByServiceId(ServiceId := pDependencies[nDependency - 1]);
			_Entries[nDependencyIndex].CompositeOwnerServiceId := _Entries[nCandidateIndex].ServiceId;
		END_FOR
		_Entries[nCandidateIndex].OwnershipState := E_CompositeOwnershipState.Owned;
	END_IF
END_FOR
END_METHOD

METHOD PUBLIC FINAL M_Register : BOOL
VAR_INPUT
	ServiceId : UDINT;
	AllowCompositeCall : BOOL;
	UpperParam : ANY;
	EffectiveParam : ANY;
END_VAR
VAR_IN_OUT
	UpperCtrl : ST_ServiceCtrl;
	EffectiveCtrl : ST_ServiceCtrl;
	Status : ST_ServiceStatus;
END_VAR
VAR
	nIndex : UINT;
	nTargetIndex : UINT;
	nUpperParamSize : UDINT;
	nEffectiveParamSize : UDINT;
	sUpperParamType : STRING(255);
	sEffectiveParamType : STRING(255);
	hrUpperParam : HRESULT;
	hrEffectiveParam : HRESULT;
END_VAR
M_Register := FALSE;
IF (_RegistrationError <> E_ServiceRegistrationError.None) OR NOT _RegistrationStarted THEN RETURN; END_IF
IF _Sealed THEN
	M_SetRegistrationError(Error := E_ServiceRegistrationError.RegistryAlreadySealed, ServiceId := ServiceId);
	RETURN;
END_IF
IF ServiceId = 0 THEN
	M_SetRegistrationError(Error := E_ServiceRegistrationError.InvalidServiceId, ServiceId := ServiceId);
	RETURN;
END_IF
FOR nIndex := 1 TO _RegisteredCount DO
	IF _Entries[nIndex].ServiceId = ServiceId THEN
		M_SetRegistrationError(Error := E_ServiceRegistrationError.DuplicateServiceId, ServiceId := ServiceId);
		RETURN;
	END_IF
END_FOR
IF _RegisteredCount >= Param_Config.MaxServicesPerModule THEN
	M_SetRegistrationError(Error := E_ServiceRegistrationError.CapacityExceeded, ServiceId := ServiceId);
	RETURN;
END_IF
IF (ADR(UpperCtrl) = 0) OR (ADR(EffectiveCtrl) = 0) OR (ADR(Status) = 0)
	OR (UpperParam.pValue = 0) OR (EffectiveParam.pValue = 0)
	OR (UpperParam.diSize <= 0) OR (EffectiveParam.diSize <= 0) THEN
	M_SetRegistrationError(Error := E_ServiceRegistrationError.InvalidStorage, ServiceId := ServiceId);
	RETURN;
END_IF
nUpperParamSize := DINT_TO_UDINT(UpperParam.diSize);
nEffectiveParamSize := DINT_TO_UDINT(EffectiveParam.diSize);
IF nUpperParamSize <> nEffectiveParamSize THEN
	M_SetRegistrationError(Error := E_ServiceRegistrationError.ParameterSizeMismatch, ServiceId := ServiceId);
	RETURN;
END_IF
sUpperParamType := _JsonDataType.GetDataTypeNameByAddress(
	nData := nUpperParamSize, pData := UpperParam.pValue, hrErrorCode => hrUpperParam);
sEffectiveParamType := _JsonDataType.GetDataTypeNameByAddress(
	nData := nEffectiveParamSize, pData := EffectiveParam.pValue, hrErrorCode => hrEffectiveParam);
IF (hrUpperParam <> 0) OR (hrEffectiveParam <> 0) OR (sUpperParamType = '') OR (sEffectiveParamType = '') THEN
	M_SetRegistrationError(Error := E_ServiceRegistrationError.ParameterTypeResolutionFailed, ServiceId := ServiceId);
	RETURN;
END_IF
IF sUpperParamType <> sEffectiveParamType THEN
	M_SetRegistrationError(Error := E_ServiceRegistrationError.ParameterTypeMismatch, ServiceId := ServiceId);
	RETURN;
END_IF
nTargetIndex := _RegisteredCount + 1;
_Entries[nTargetIndex].InUse := TRUE;
_Entries[nTargetIndex].ServiceId := ServiceId;
_Entries[nTargetIndex].AllowCompositeCall := AllowCompositeCall;
_Entries[nTargetIndex].UpperCtrlAddress := ADR(UpperCtrl);
_Entries[nTargetIndex].EffectiveCtrlAddress := ADR(EffectiveCtrl);
_Entries[nTargetIndex].UpperParamAddress := UpperParam.pValue;
_Entries[nTargetIndex].EffectiveParamAddress := EffectiveParam.pValue;
_Entries[nTargetIndex].ParameterSize := nUpperParamSize;
_Entries[nTargetIndex].ParameterTypeName := sUpperParamType;
_Entries[nTargetIndex].StatusAddress := ADR(Status);
_Entries[nTargetIndex].InternalCommandState := E_ServiceInternalCommandState.None;
_Entries[nTargetIndex].OwnershipState := E_CompositeOwnershipState.None;
_RegisteredCount := nTargetIndex;
M_Register := TRUE;
END_METHOD

METHOD PUBLIC FINAL M_RegisterCompositeDefinition : BOOL
VAR_INPUT
	CompositeServiceId : UDINT;
	DependencyCount : UINT;
END_VAR
VAR_IN_OUT
	DependencyIds : ARRAY[1..Param_Config.MaxCompositeDependencies] OF UDINT;
END_VAR
VAR
	nCompositeIndex : UINT;
	nDependencyIndex : UINT;
	nDependency : UINT;
	nOtherDependency : UINT;
END_VAR
M_RegisterCompositeDefinition := FALSE;
IF (_RegistrationError <> E_ServiceRegistrationError.None) OR NOT _RegistrationStarted THEN RETURN; END_IF
IF _Sealed THEN
	M_SetRegistrationError(Error := E_ServiceRegistrationError.RegistryAlreadySealed, ServiceId := CompositeServiceId);
	RETURN;
END_IF
nCompositeIndex := M_FindIndexByServiceId(ServiceId := CompositeServiceId);
IF nCompositeIndex = 0 THEN
	M_SetRegistrationError(Error := E_ServiceRegistrationError.InvalidCompositeService, ServiceId := CompositeServiceId);
	RETURN;
END_IF
IF _Entries[nCompositeIndex].IsComposite THEN
	M_SetRegistrationError(Error := E_ServiceRegistrationError.DuplicateCompositeDefinition, ServiceId := CompositeServiceId);
	RETURN;
END_IF
IF DependencyCount = 0 THEN
	M_SetRegistrationError(Error := E_ServiceRegistrationError.EmptyCompositeDependencyList, ServiceId := CompositeServiceId);
	RETURN;
END_IF
IF DependencyCount > Param_Config.MaxCompositeDependencies THEN
	M_SetRegistrationError(Error := E_ServiceRegistrationError.CompositeDependencyCapacityExceeded, ServiceId := CompositeServiceId);
	RETURN;
END_IF
FOR nDependency := 1 TO DependencyCount DO
	IF DependencyIds[nDependency] = 0 THEN
		M_SetRegistrationError(Error := E_ServiceRegistrationError.InvalidCompositeDependencyId, ServiceId := CompositeServiceId);
		RETURN;
	END_IF
	IF DependencyIds[nDependency] = CompositeServiceId THEN
		M_SetRegistrationError(Error := E_ServiceRegistrationError.SelfDependency, ServiceId := CompositeServiceId);
		RETURN;
	END_IF
	nDependencyIndex := M_FindIndexByServiceId(ServiceId := DependencyIds[nDependency]);
	IF nDependencyIndex = 0 THEN
		M_SetRegistrationError(Error := E_ServiceRegistrationError.UnknownCompositeDependency, ServiceId := DependencyIds[nDependency]);
		RETURN;
	END_IF
	IF NOT _Entries[nDependencyIndex].AllowCompositeCall THEN
		M_SetRegistrationError(Error := E_ServiceRegistrationError.CompositeDependencyNotAllowed, ServiceId := DependencyIds[nDependency]);
		RETURN;
	END_IF
	FOR nOtherDependency := 1 TO nDependency - 1 DO
		IF DependencyIds[nOtherDependency] = DependencyIds[nDependency] THEN
			M_SetRegistrationError(Error := E_ServiceRegistrationError.DuplicateCompositeDependency, ServiceId := DependencyIds[nDependency]);
			RETURN;
		END_IF
	END_FOR
END_FOR
_Entries[nCompositeIndex].IsComposite := TRUE;
_Entries[nCompositeIndex].CompositeDependenciesAddress := ADR(DependencyIds);
_Entries[nCompositeIndex].CompositeDependencyCount := DependencyCount;
_Entries[nCompositeIndex].OwnershipState := E_CompositeOwnershipState.None;
M_RegisterCompositeDefinition := TRUE;
END_METHOD

METHOD PUBLIC FINAL M_ReleaseCompositeOwnership : BOOL
VAR_INPUT
	CompositeServiceId : UDINT;
END_VAR
VAR
	nCompositeIndex : UINT;
	nDependencyIndex : UINT;
	nDependency : UINT;
	pDependencies : POINTER TO UDINT;
	pEffectiveCtrl : POINTER TO ST_ServiceCtrl;
END_VAR
M_ReleaseCompositeOwnership := FALSE;
nCompositeIndex := M_FindIndexByServiceId(ServiceId := CompositeServiceId);
IF (nCompositeIndex = 0) OR NOT _Entries[nCompositeIndex].IsComposite THEN RETURN; END_IF
pDependencies := _Entries[nCompositeIndex].CompositeDependenciesAddress;
FOR nDependency := 1 TO _Entries[nCompositeIndex].CompositeDependencyCount DO
	nDependencyIndex := M_FindIndexByServiceId(ServiceId := pDependencies[nDependency - 1]);
	IF _Entries[nDependencyIndex].CompositeOwnerServiceId = CompositeServiceId THEN
		_Entries[nDependencyIndex].CompositeOwnerServiceId := 0;
		IF (_Entries[nDependencyIndex].InternalCommandState = E_ServiceInternalCommandState.Queued)
			OR (_Entries[nDependencyIndex].InternalCommandState = E_ServiceInternalCommandState.RequestHigh) THEN
			_Entries[nDependencyIndex].InternalCommandState := E_ServiceInternalCommandState.Cancelled;
		END_IF
		_Entries[nDependencyIndex].InternalRequestMustGoLow := FALSE;
		pEffectiveCtrl := _Entries[nDependencyIndex].EffectiveCtrlAddress;
		pEffectiveCtrl^.PackMLIn.bCommandChangeRequest := FALSE;
	END_IF
END_FOR
_Entries[nCompositeIndex].OwnershipState := E_CompositeOwnershipState.None;
M_ReleaseCompositeOwnership := TRUE;
END_METHOD

METHOD PUBLIC FINAL M_RequestCompositeOwnership : BOOL
VAR_INPUT
	CompositeServiceId : UDINT;
END_VAR
VAR
	nIndex : UINT;
END_VAR
M_RequestCompositeOwnership := FALSE;
IF NOT Ready THEN RETURN; END_IF
nIndex := M_FindIndexByServiceId(ServiceId := CompositeServiceId);
IF (nIndex = 0) OR NOT _Entries[nIndex].IsComposite THEN RETURN; END_IF
IF _Entries[nIndex].OwnershipState = E_CompositeOwnershipState.Owned THEN
	M_RequestCompositeOwnership := TRUE;
	RETURN;
END_IF
_Entries[nIndex].OwnershipState := E_CompositeOwnershipState.Pending;
M_RequestCompositeOwnership := TRUE;
END_METHOD

METHOD PUBLIC FINAL M_Seal : BOOL
VAR
	nIndex : UINT;
	nDependency : UINT;
	nDependencyIndex : UINT;
	pDependencies : POINTER TO UDINT;
	pEffectiveCtrl : POINTER TO ST_ServiceCtrl;
END_VAR
M_Seal := FALSE;
IF _RegistrationError <> E_ServiceRegistrationError.None THEN RETURN; END_IF
IF _Sealed THEN
	M_SetRegistrationError(Error := E_ServiceRegistrationError.RegistryAlreadySealed, ServiceId := 0);
	RETURN;
END_IF
IF NOT _RegistrationStarted OR (_RegisteredCount = 0) THEN
	M_SetRegistrationError(Error := E_ServiceRegistrationError.EmptyRegistry, ServiceId := 0);
	RETURN;
END_IF
FOR nIndex := 1 TO _RegisteredCount DO
	IF _Entries[nIndex].IsComposite THEN
		pDependencies := _Entries[nIndex].CompositeDependenciesAddress;
		FOR nDependency := 1 TO _Entries[nIndex].CompositeDependencyCount DO
			nDependencyIndex := M_FindIndexByServiceId(ServiceId := pDependencies[nDependency - 1]);
			IF _Entries[nDependencyIndex].IsComposite THEN
				M_SetRegistrationError(Error := E_ServiceRegistrationError.NestedCompositeNotSupported,
					ServiceId := _Entries[nDependencyIndex].ServiceId);
				RETURN;
			END_IF
		END_FOR
	END_IF
END_FOR
FOR nIndex := 1 TO _RegisteredCount DO
	pEffectiveCtrl := _Entries[nIndex].EffectiveCtrlAddress;
	pEffectiveCtrl^.PackMLIn.bCommandChangeRequest := FALSE;
	pEffectiveCtrl^.PackMLIn.bModeChangeRequest := FALSE;
	_Entries[nIndex].ObservedSnapshot.Valid := FALSE;
END_FOR
_AllIdle := FALSE;
_AllStopped := FALSE;
_AllAborted := FALSE;
_Sealed := TRUE;
M_Seal := TRUE;
END_METHOD

METHOD PRIVATE M_SetRegistrationError
VAR_INPUT
	Error : E_ServiceRegistrationError;
	ServiceId : UDINT;
END_VAR
IF _RegistrationError <> E_ServiceRegistrationError.None THEN RETURN; END_IF
_RegistrationError := Error;
_FailedServiceId := ServiceId;
_Sealed := FALSE;
_AllIdle := FALSE;
_AllStopped := FALSE;
_AllAborted := FALSE;
END_METHOD

METHOD PUBLIC FINAL M_SubmitInternalCommand : E_ServiceCallSubmitResult
VAR_INPUT
	CallerServiceId : UDINT;
	TargetServiceId : UDINT;
	RequestId : UDINT;
	Command : E_PackMLCommand;
END_VAR
VAR
	nCallerIndex : UINT;
	nTargetIndex : UINT;
END_VAR
IF NOT Ready THEN
	M_SubmitInternalCommand := E_ServiceCallSubmitResult.CoordinatorNotReady;
	RETURN;
END_IF

// Accept ONLY Stop, Abort, Clear, Reset cmd
IF (Command <> E_PackMLCommand.Stop) AND (Command <> E_PackMLCommand.Abort)
	AND (Command <> E_PackMLCommand.Clear) AND (Command <> E_PackMLCommand.Reset) THEN
	M_SubmitInternalCommand := E_ServiceCallSubmitResult.InvalidCommand;
	RETURN;
END_IF

nTargetIndex := M_FindIndexByServiceId(ServiceId := TargetServiceId);
IF nTargetIndex = 0 THEN
	M_SubmitInternalCommand := E_ServiceCallSubmitResult.UnknownService;
	RETURN;
END_IF

nCallerIndex := M_FindIndexByServiceId(ServiceId := CallerServiceId);
IF (nCallerIndex = 0) OR NOT M_IsDeclaredDependency(
	CompositeIndex := nCallerIndex, TargetServiceId := TargetServiceId) THEN
	M_SubmitInternalCommand := E_ServiceCallSubmitResult.DependencyNotDeclared;
	RETURN;
END_IF
IF _Entries[nTargetIndex].CompositeOwnerServiceId <> CallerServiceId THEN
	M_SubmitInternalCommand := E_ServiceCallSubmitResult.NotOwner;
	RETURN;
END_IF
IF (_Entries[nTargetIndex].InternalCommandState = E_ServiceInternalCommandState.Queued)
	OR (_Entries[nTargetIndex].InternalCommandState = E_ServiceInternalCommandState.RequestHigh)
	OR _Entries[nTargetIndex].InternalRequestMustGoLow THEN
	M_SubmitInternalCommand := E_ServiceCallSubmitResult.Busy;
	RETURN;
END_IF
_Entries[nTargetIndex].InternalRequestId := RequestId;
_Entries[nTargetIndex].InternalCommand := Command;
_Entries[nTargetIndex].InternalCommandState := E_ServiceInternalCommandState.Queued;
_Entries[nTargetIndex].InternalRequestMustGoLow := FALSE;
M_SubmitInternalCommand := E_ServiceCallSubmitResult.Queued;
END_METHOD

METHOD PUBLIC FINAL M_SubmitInternalStart : E_ServiceCallSubmitResult
VAR_INPUT
	CallerServiceId : UDINT;
	TargetServiceId : UDINT;
	RequestId : UDINT;
	Parameters : ANY;
END_VAR
VAR
	nCallerIndex : UINT;
	nTargetIndex : UINT;
	nParameterSize : UDINT;
	sParameterType : STRING(255);
	hrParameter : HRESULT;
END_VAR
IF NOT Ready THEN
	M_SubmitInternalStart := E_ServiceCallSubmitResult.CoordinatorNotReady;
	RETURN;
END_IF
nTargetIndex := M_FindIndexByServiceId(ServiceId := TargetServiceId);
IF nTargetIndex = 0 THEN
	M_SubmitInternalStart := E_ServiceCallSubmitResult.UnknownService;
	RETURN;
END_IF
nCallerIndex := M_FindIndexByServiceId(ServiceId := CallerServiceId);
IF (nCallerIndex = 0) OR NOT M_IsDeclaredDependency(
	CompositeIndex := nCallerIndex, TargetServiceId := TargetServiceId) THEN
	M_SubmitInternalStart := E_ServiceCallSubmitResult.DependencyNotDeclared;
	RETURN;
END_IF
IF _Entries[nTargetIndex].CompositeOwnerServiceId <> CallerServiceId THEN
	M_SubmitInternalStart := E_ServiceCallSubmitResult.NotOwner;
	RETURN;
END_IF
IF (_Entries[nTargetIndex].InternalCommandState = E_ServiceInternalCommandState.Queued)
	OR (_Entries[nTargetIndex].InternalCommandState = E_ServiceInternalCommandState.RequestHigh)
	OR _Entries[nTargetIndex].InternalRequestMustGoLow THEN
	M_SubmitInternalStart := E_ServiceCallSubmitResult.Busy;
	RETURN;
END_IF
IF (Parameters.pValue = 0) OR (Parameters.diSize <= 0) THEN
	M_SubmitInternalStart := E_ServiceCallSubmitResult.ParameterSizeMismatch;
	RETURN;
END_IF
nParameterSize := DINT_TO_UDINT(Parameters.diSize);
IF nParameterSize <> _Entries[nTargetIndex].ParameterSize THEN
	M_SubmitInternalStart := E_ServiceCallSubmitResult.ParameterSizeMismatch;
	RETURN;
END_IF
sParameterType := _JsonDataType.GetDataTypeNameByAddress(
	nData := nParameterSize, pData := Parameters.pValue, hrErrorCode => hrParameter);
IF (hrParameter <> 0) OR (sParameterType = '') THEN
	M_SubmitInternalStart := E_ServiceCallSubmitResult.ParameterTypeResolutionFailed;
	RETURN;
END_IF
IF sParameterType <> _Entries[nTargetIndex].ParameterTypeName THEN
	M_SubmitInternalStart := E_ServiceCallSubmitResult.ParameterTypeMismatch;
	RETURN;
END_IF
MEMCPY(destAddr := _Entries[nTargetIndex].EffectiveParamAddress,
	srcAddr := Parameters.pValue, n := nParameterSize);
_Entries[nTargetIndex].InternalRequestId := RequestId;
_Entries[nTargetIndex].InternalCommand := E_PackMLCommand.Start;
_Entries[nTargetIndex].InternalCommandState := E_ServiceInternalCommandState.Queued;
_Entries[nTargetIndex].InternalRequestMustGoLow := FALSE;
M_SubmitInternalStart := E_ServiceCallSubmitResult.Queued;
END_METHOD

PROPERTY PUBLIC FINAL Ready : BOOL
GET
Ready := _RegistrationStarted AND _Sealed
	AND (_RegistrationError = E_ServiceRegistrationError.None);
END_GET
END_PROPERTY

PROPERTY PUBLIC FINAL RegisteredCount : UINT
GET
RegisteredCount := _RegisteredCount;
END_GET
END_PROPERTY

PROPERTY PUBLIC FINAL RegistrationError : E_ServiceRegistrationError
GET
RegistrationError := _RegistrationError;
END_GET
END_PROPERTY

END_FUNCTION_BLOCK

// ---- POUs/10_Module/FB_ServiceCaller.TcPOU
FUNCTION_BLOCK FB_ServiceCaller
VAR
	_Coordinator : REFERENCE TO FB_ServiceCoordinator;
	_CallerServiceId : UDINT;
	_NextRequestId : UDINT;
	_Configured : BOOL;
END_VAR

METHOD PUBLIC FINAL M_Command : E_ServiceCallSubmitResult
VAR_INPUT
	ServiceId : UDINT;
	Command : E_PackMLCommand;
END_VAR
VAR
	nRequestId : UDINT;
END_VAR
IF NOT _Configured OR NOT __ISVALIDREF(_Coordinator) THEN
	M_Command := E_ServiceCallSubmitResult.CallerNotConfigured;
	RETURN;
END_IF
nRequestId := _NextRequestId + 1;
IF nRequestId = 0 THEN nRequestId := 1; END_IF
M_Command := _Coordinator.M_SubmitInternalCommand(
	CallerServiceId := _CallerServiceId,
	TargetServiceId := ServiceId,
	RequestId := nRequestId,
	Command := Command);
IF M_Command = E_ServiceCallSubmitResult.Queued THEN
	_NextRequestId := nRequestId;
END_IF
END_METHOD

METHOD PUBLIC FINAL M_Configure : BOOL
VAR_INPUT
	CallerServiceId : UDINT;
END_VAR
VAR_IN_OUT
	Coordinator : FB_ServiceCoordinator;
END_VAR
M_Configure := FALSE;
IF CallerServiceId = 0 THEN RETURN; END_IF
_Coordinator REF= Coordinator;
_CallerServiceId := CallerServiceId;
_NextRequestId := 0;
_Configured := TRUE;
M_Configure := TRUE;
END_METHOD

METHOD PUBLIC FINAL M_GetCommandState : E_ServiceInternalCommandState
VAR_INPUT
	ServiceId : UDINT;
END_VAR
M_GetCommandState := E_ServiceInternalCommandState.None;
IF NOT _Configured OR NOT __ISVALIDREF(_Coordinator) THEN RETURN; END_IF
M_GetCommandState := _Coordinator.M_GetInternalCommandState(
	CallerServiceId := _CallerServiceId,
	TargetServiceId := ServiceId);
END_METHOD

METHOD PUBLIC FINAL M_GetServiceSnapshot : BOOL
VAR_INPUT
	ServiceId : UDINT;
END_VAR
VAR_OUTPUT
	Snapshot : ST_ServiceExecutionSnapshot;
END_VAR
M_GetServiceSnapshot := FALSE;
MEMSET(ADR(Snapshot), 0, SIZEOF(Snapshot));
IF NOT _Configured OR NOT __ISVALIDREF(_Coordinator) THEN RETURN; END_IF
M_GetServiceSnapshot := _Coordinator.M_GetServiceSnapshotById(
	ServiceId := ServiceId,
	Snapshot => Snapshot);
END_METHOD

METHOD PUBLIC FINAL M_Start : E_ServiceCallSubmitResult
VAR_INPUT
	ServiceId : UDINT;
	Parameters : ANY;
END_VAR
VAR
	nRequestId : UDINT;
END_VAR
IF NOT _Configured OR NOT __ISVALIDREF(_Coordinator) THEN
	M_Start := E_ServiceCallSubmitResult.CallerNotConfigured;
	RETURN;
END_IF
nRequestId := _NextRequestId + 1;
IF nRequestId = 0 THEN nRequestId := 1; END_IF
M_Start := _Coordinator.M_SubmitInternalStart(
	CallerServiceId := _CallerServiceId,
	TargetServiceId := ServiceId,
	RequestId := nRequestId,
	Parameters := Parameters);
IF M_Start = E_ServiceCallSubmitResult.Queued THEN
	_NextRequestId := nRequestId;
END_IF
END_METHOD

END_FUNCTION_BLOCK

// ---- POUs/30_PackML_Base/FB_PackMLBase.TcPOU
FUNCTION_BLOCK FB_PackMLBase
VAR_INPUT
	PackMLIn	: ST_PML_Base_In;
	
	bEnable				: BOOL := TRUE;
	bExternalFault		: BOOL;
END_VAR
VAR_OUTPUT
	PackMLOut	: ST_PML_Base_Out;
	
	bTransitionActive	: BOOL;
END_VAR
VAR
	_eLastCommand			: E_PackMLCommand := E_PackMLCommand.None;
	_eCommandToProcess		: E_PackMLCommand := E_PackMLCommand.None;
	_eQueuedCommand			: E_PackMLCommand := E_PackMLCommand.None;
	_bQueuedCommandRequest	: BOOL;
	_bCommandConsumed		: BOOL;
	_bModeChangeConsumed	: BOOL;
	_bStateFirstScan		: BOOL := TRUE;
	_bStateFirstScanForHook	: BOOL;
	_eHookResult			: E_PackMLHookResult;
END_VAR

// Reset edge-style status before evaluating this PLC cycle.
_eCommandToProcess		:= E_PackMLCommand.None;

// Command and mode request feedback is latched for HMI/upper-layer handshakes
// until the corresponding request input returns to FALSE.
IF NOT PackMLIn.bCommandChangeRequest THEN
	PackMLOut.bCommandAccepted	:= FALSE;
	PackMLOut.bCommandRejected	:= FALSE;
	PackMLOut.eStateErrorID			:= E_PackMLErrorID.NoError;
END_IF

IF NOT PackMLIn.bModeChangeRequest THEN
	PackMLOut.bModeChanged		:= FALSE;
	PackMLOut.bModeChangeRejected	:= FALSE;
	PackMLOut.eModeErrorID		:= E_PackMLErrorID.NoError;
END_IF

// A disabled base FB holds the current state and suppresses transition activity.
IF NOT bEnable THEN
	bTransitionActive := FALSE;
	RETURN;
END_IF

// Mode change requests are edge/latch based, matching command request behavior.
// The caller must clear stIn.bModeChangeRequest before the same request can run again.
IF NOT PackMLIn.bModeChangeRequest THEN
	_bModeChangeConsumed := FALSE;
END_IF

IF PackMLIn.bModeChangeRequest AND NOT _bModeChangeConsumed THEN
	_bModeChangeConsumed := TRUE;

	IF NOT H_IsModeSupported(PackMLIn.eMode) THEN
		M_RejectModeChange(E_PackMLErrorID.ModeNotSupported);
	ELSIF PackMLIn.eMode = PackMLOut.eModeCurrent THEN
		M_RejectModeChange(E_PackMLErrorID.ModeAlreadyActive);
	ELSIF NOT M_IsModeChangeAllowedByState() THEN
		M_RejectModeChange(E_PackMLErrorID.ModeChangeNotAllowedFromCurrentState);
	ELSIF NOT H_IsStateSupportedByMode(PackMLIn.eMode, PackMLOut.eStateCurrent) THEN
		M_RejectModeChange(E_PackMLErrorID.ModeDoesNotSupportCurrentState);
	ELSE
		M_ChangeMode(PackMLIn.eMode);
	END_IF
END_IF

// Command requests are edge/latch based, matching mode-change request behavior.
// The caller must clear stIn.bCommandChangeRequest before another command can run.
IF NOT PackMLIn.bCommandChangeRequest THEN
	_bCommandConsumed	:= FALSE;
	_eLastCommand		:= E_PackMLCommand.None;
END_IF

// External faults have priority over normal commands and force the abort path
// only while the machine is not already Aborting or Aborted.
IF bExternalFault AND M_IsAbortAllowedByState() THEN
	_eCommandToProcess := E_PackMLCommand.Abort;
ELSIF _bQueuedCommandRequest AND (_eQueuedCommand <> E_PackMLCommand.None) THEN
	_eCommandToProcess		:= _eQueuedCommand;
	_eQueuedCommand			:= E_PackMLCommand.None;
	_bQueuedCommandRequest	:= FALSE;
ELSIF PackMLIn.bCommandChangeRequest AND (PackMLIn.eCommand <> E_PackMLCommand.None) AND NOT _bCommandConsumed THEN
	_eCommandToProcess	:= PackMLIn.eCommand;
	_eLastCommand		:= PackMLIn.eCommand;
	_bCommandConsumed	:= TRUE;
END_IF

// Mode policy hooks run before PackML state guards so a forbidden command reports
// the mode reason instead of a state reason.
IF (_eCommandToProcess <> E_PackMLCommand.None) AND NOT H_IsCommandAllowedByMode(_eCommandToProcess, PackMLOut.eModeCurrent) THEN
	M_RejectCommand(E_PackMLErrorID.CommandNotAllowedInActiveMode);
	_eCommandToProcess := E_PackMLCommand.None;
END_IF

// Dispatch the accepted command through private PackML state guards.
// Rejected commands never mutate the state and return a stable numeric error ID.
CASE _eCommandToProcess OF
	E_PackMLCommand.Clear:
		IF M_IsClearAllowedByState() THEN
			PackMLOut.bCommandAccepted := TRUE;
			M_ChangeState(E_PackMLState.Clearing);
		ELSE
			M_RejectCommand(E_PackMLErrorID.ClearNotAllowedFromCurrentState);
		END_IF

	E_PackMLCommand.Reset:
		IF M_IsResetAllowedByState() THEN
			PackMLOut.bCommandAccepted := TRUE;
			M_ChangeState(E_PackMLState.Resetting);
		ELSE
			M_RejectCommand(E_PackMLErrorID.ResetNotAllowedFromCurrentState);
		END_IF

	E_PackMLCommand.Start:
		IF M_IsStartAllowedByState() THEN
			PackMLOut.bCommandAccepted := TRUE;
			M_ChangeState(E_PackMLState.Starting);
		ELSE
			M_RejectCommand(E_PackMLErrorID.StartNotAllowedFromCurrentState);
		END_IF

	E_PackMLCommand.Stop:
		IF M_IsStopAllowedByState() THEN
			PackMLOut.bCommandAccepted := TRUE;
			M_ChangeState(E_PackMLState.Stopping);
		ELSE
			M_RejectCommand(E_PackMLErrorID.StopNotAllowedFromCurrentState);
		END_IF

	E_PackMLCommand.Hold:
		IF M_IsHoldAllowedByState() THEN
			PackMLOut.bCommandAccepted := TRUE;
			M_ChangeState(E_PackMLState.Holding);
		ELSE
			M_RejectCommand(E_PackMLErrorID.HoldNotAllowedFromCurrentState);
		END_IF

	E_PackMLCommand.Unhold:
		IF M_IsUnholdAllowedByState() THEN
			PackMLOut.bCommandAccepted := TRUE;
			M_ChangeState(E_PackMLState.Unholding);
		ELSE
			M_RejectCommand(E_PackMLErrorID.UnholdNotAllowedFromCurrentState);
		END_IF

	E_PackMLCommand.Suspend:
		IF M_IsSuspendAllowedByState() THEN
			PackMLOut.bCommandAccepted := TRUE;
			M_ChangeState(E_PackMLState.Suspending);
		ELSE
			M_RejectCommand(E_PackMLErrorID.SuspendNotAllowedFromCurrentState);
		END_IF

	E_PackMLCommand.Unsuspend:
		IF M_IsUnsuspendAllowedByState() THEN
			PackMLOut.bCommandAccepted := TRUE;
			M_ChangeState(E_PackMLState.Unsuspending);
		ELSE
			M_RejectCommand(E_PackMLErrorID.UnsuspendNotAllowedFromCurrentState);
		END_IF

	E_PackMLCommand.Abort:
		IF M_IsAbortAllowedByState() THEN
			PackMLOut.bCommandAccepted := TRUE;
			M_ChangeState(E_PackMLState.Aborting);
		ELSE
			M_RejectCommand(E_PackMLErrorID.AbortNotAllowedFromCurrentState);
		END_IF
END_CASE

// Run the current state's action hook, then advance transient states when their
// hook reports Done. Stable states remain active until a command moves them.
_bStateFirstScanForHook	:= _bStateFirstScan;
_bStateFirstScan		:= FALSE;

CASE PackMLOut.eStateCurrent OF
	E_PackMLState.Undefined:
		_eHookResult := H_OnUndefined(_bStateFirstScanForHook);
		IF _eHookResult = E_PackMLHookResult.Done THEN
			M_ChangeState(E_PackMLState.Aborted);
		END_IF

	E_PackMLState.Clearing:
		_eHookResult := H_OnClearing(_bStateFirstScanForHook);
		IF _eHookResult = E_PackMLHookResult.Done THEN
			M_ChangeState(E_PackMLState.Stopped);
		END_IF

	E_PackMLState.Stopped:
		H_OnStopped(_bStateFirstScanForHook);

	E_PackMLState.Starting:
		_eHookResult := H_OnStarting(_bStateFirstScanForHook);
		IF _eHookResult = E_PackMLHookResult.Done THEN
			M_ChangeState(E_PackMLState.Execute);
		END_IF

	E_PackMLState.Idle:
		H_OnIdle(_bStateFirstScanForHook);

	E_PackMLState.Suspended:
		H_OnSuspended(_bStateFirstScanForHook);

	E_PackMLState.Execute:
		_eHookResult := H_OnExecute(_bStateFirstScanForHook);
		IF _eHookResult = E_PackMLHookResult.Done THEN
			M_ChangeState(E_PackMLState.Completing);
		END_IF

	E_PackMLState.Stopping:
		_eHookResult := H_OnStopping(_bStateFirstScanForHook);
		IF _eHookResult = E_PackMLHookResult.Done THEN
			M_ChangeState(E_PackMLState.Stopped);
		END_IF

	E_PackMLState.Aborting:
		_eHookResult := H_OnAborting(_bStateFirstScanForHook);
		IF _eHookResult = E_PackMLHookResult.Done THEN
			M_ChangeState(E_PackMLState.Aborted);
		END_IF

	E_PackMLState.Aborted:
		H_OnAborted(_bStateFirstScanForHook);

	E_PackMLState.Holding:
		_eHookResult := H_OnHolding(_bStateFirstScanForHook);
		IF _eHookResult = E_PackMLHookResult.Done THEN
			M_ChangeState(E_PackMLState.Held);
		END_IF

	E_PackMLState.Held:
		H_OnHeld(_bStateFirstScanForHook);

	E_PackMLState.Unholding:
		_eHookResult := H_OnUnholding(_bStateFirstScanForHook);
		IF _eHookResult = E_PackMLHookResult.Done THEN
			M_ChangeState(E_PackMLState.Execute);
		END_IF

	E_PackMLState.Suspending:
		_eHookResult := H_OnSuspending(_bStateFirstScanForHook);
		IF _eHookResult = E_PackMLHookResult.Done THEN
			M_ChangeState(E_PackMLState.Suspended);
		END_IF

	E_PackMLState.Unsuspending:
		_eHookResult := H_OnUnsuspending(_bStateFirstScanForHook);
		IF _eHookResult = E_PackMLHookResult.Done THEN
			M_ChangeState(E_PackMLState.Execute);
		END_IF

	E_PackMLState.Resetting:
		_eHookResult := H_OnResetting(_bStateFirstScanForHook);
		IF _eHookResult = E_PackMLHookResult.Done THEN
			M_ChangeState(E_PackMLState.Idle);
		END_IF

	E_PackMLState.Completing:
		_eHookResult := H_OnCompleting(_bStateFirstScanForHook);
		IF _eHookResult = E_PackMLHookResult.Done THEN
			M_ChangeState(E_PackMLState.Complete);
		END_IF

	E_PackMLState.Complete:
		H_OnComplete(_bStateFirstScanForHook);
END_CASE

// Transition activity is true for transient states that normally need completion
// confirmation from their state hook.
bTransitionActive :=
	(PackMLOut.eStateCurrent = E_PackMLState.Undefined) OR
	(PackMLOut.eStateCurrent = E_PackMLState.Clearing) OR
	(PackMLOut.eStateCurrent = E_PackMLState.Starting) OR
	(PackMLOut.eStateCurrent = E_PackMLState.Stopping) OR
	(PackMLOut.eStateCurrent = E_PackMLState.Aborting) OR
	(PackMLOut.eStateCurrent = E_PackMLState.Holding) OR
	(PackMLOut.eStateCurrent = E_PackMLState.Unholding) OR
	(PackMLOut.eStateCurrent = E_PackMLState.Suspending) OR
	(PackMLOut.eStateCurrent = E_PackMLState.Unsuspending) OR
	(PackMLOut.eStateCurrent = E_PackMLState.Resetting) OR
	(PackMLOut.eStateCurrent = E_PackMLState.Completing);

METHOD PROTECTED H_IsCommandAllowedByMode : BOOL
VAR_INPUT
	eRequestedCommand	: E_PackMLCommand;
	eActiveMode			: T_PackMLMode;
END_VAR
// Modes are application-defined in library use; override to restrict commands per mode.
H_IsCommandAllowedByMode := TRUE;
END_METHOD

METHOD PROTECTED H_IsModeSupported : BOOL
VAR_INPUT
	eRequestedMode	: T_PackMLMode;
END_VAR
// Modes are application-defined in library use; override to reject unsupported modes.
H_IsModeSupported := TRUE;
END_METHOD

METHOD PROTECTED H_IsStateSupportedByMode : BOOL
VAR_INPUT
	eRequestedMode	: T_PackMLMode;
	eCurrentState	: E_PackMLState;
END_VAR
// Modes are application-defined in library use; override to restrict mode/state pairs.
H_IsStateSupportedByMode := TRUE;
END_METHOD

METHOD PROTECTED H_OnAborted
VAR_INPUT
	bFirstScan	: BOOL;
END_VAR
// Default action hook intentionally empty. Override in derived FBs when needed.
END_METHOD

METHOD PROTECTED H_OnAborting : E_PackMLHookResult
VAR_INPUT
	bFirstScan	: BOOL;
END_VAR
// Default transient hooks complete immediately; override when work is required.
H_OnAborting := E_PackMLHookResult.Done;
END_METHOD

METHOD PROTECTED H_OnClearing : E_PackMLHookResult
VAR_INPUT
	bFirstScan	: BOOL;
END_VAR
// Default transient hooks complete immediately; override when work is required.
H_OnClearing := E_PackMLHookResult.Done;
END_METHOD

METHOD PROTECTED H_OnComplete
VAR_INPUT
	bFirstScan	: BOOL;
END_VAR
// Default action hook intentionally empty. Override in derived FBs when needed.
END_METHOD

METHOD PROTECTED H_OnCompleting : E_PackMLHookResult
VAR_INPUT
	bFirstScan	: BOOL;
END_VAR
// Default transient hooks complete immediately; override when work is required.
H_OnCompleting := E_PackMLHookResult.Done;
END_METHOD

METHOD PROTECTED H_OnExecute : E_PackMLHookResult
VAR_INPUT
	bFirstScan	: BOOL;
END_VAR
// Execute is stable by default; derived FBs decide when the process is done.
H_OnExecute := E_PackMLHookResult.Busy;
END_METHOD

METHOD PROTECTED H_OnHeld
VAR_INPUT
	bFirstScan	: BOOL;
END_VAR
// Default action hook intentionally empty. Override in derived FBs when needed.
END_METHOD

METHOD PROTECTED H_OnHolding : E_PackMLHookResult
VAR_INPUT
	bFirstScan	: BOOL;
END_VAR
// Default transient hooks complete immediately; override when work is required.
H_OnHolding := E_PackMLHookResult.Done;
END_METHOD

METHOD PROTECTED H_OnIdle
VAR_INPUT
	bFirstScan	: BOOL;
END_VAR
// Default action hook intentionally empty. Override in derived FBs when needed.
END_METHOD

METHOD PROTECTED H_OnModeChanged
VAR_INPUT
	ePreviousMode	: T_PackMLMode;
	eNewMode		: T_PackMLMode;
END_VAR
// Default mode-change hook intentionally empty. Override in derived FBs when needed.
END_METHOD

METHOD PROTECTED H_OnResetting : E_PackMLHookResult
VAR_INPUT
	bFirstScan	: BOOL;
END_VAR
// Default transient hooks complete immediately; override when work is required.
H_OnResetting := E_PackMLHookResult.Done;
END_METHOD

METHOD PROTECTED H_OnStarting : E_PackMLHookResult
VAR_INPUT
	bFirstScan	: BOOL;
END_VAR
// Default transient hooks complete immediately; override when work is required.
H_OnStarting := E_PackMLHookResult.Done;
END_METHOD

METHOD PROTECTED H_OnStateChanged
VAR_INPUT
	ePreviousState	: E_PackMLState;
	eNewState		: E_PackMLState;
END_VAR
// Default state-change hook intentionally empty. Override in derived FBs when needed.
END_METHOD

METHOD PROTECTED H_OnStopped
VAR_INPUT
	bFirstScan	: BOOL;
END_VAR
// Default action hook intentionally empty. Override in derived FBs when needed.
END_METHOD

METHOD PROTECTED H_OnStopping : E_PackMLHookResult
VAR_INPUT
	bFirstScan	: BOOL;
END_VAR
// Default transient hooks complete immediately; override when work is required.
H_OnStopping := E_PackMLHookResult.Done;
END_METHOD

METHOD PROTECTED H_OnSuspended
VAR_INPUT
	bFirstScan	: BOOL;
END_VAR
// Default action hook intentionally empty. Override in derived FBs when needed.
END_METHOD

METHOD PROTECTED H_OnSuspending : E_PackMLHookResult
VAR_INPUT
	bFirstScan	: BOOL;
END_VAR
// Default transient hooks complete immediately; override when work is required.
H_OnSuspending := E_PackMLHookResult.Done;
END_METHOD

METHOD PROTECTED H_OnUndefined : E_PackMLHookResult
VAR_INPUT
	bFirstScan	: BOOL;
END_VAR
// The base FB leaves Undefined immediately unless a derived FB delays startup.
H_OnUndefined := E_PackMLHookResult.Done;
END_METHOD

METHOD PROTECTED H_OnUnholding : E_PackMLHookResult
VAR_INPUT
	bFirstScan	: BOOL;
END_VAR
// Default transient hooks complete immediately; override when work is required.
H_OnUnholding := E_PackMLHookResult.Done;
END_METHOD

METHOD PROTECTED H_OnUnsuspending : E_PackMLHookResult
VAR_INPUT
	bFirstScan	: BOOL;
END_VAR
// Default transient hooks complete immediately; override when work is required.
H_OnUnsuspending := E_PackMLHookResult.Done;
END_METHOD

METHOD PRIVATE M_ChangeMode
VAR_INPUT
	eNextMode	: T_PackMLMode;
END_VAR
// Centralize mode mutation so previous-mode and edge outputs stay consistent.
IF PackMLOut.eModeCurrent <> eNextMode THEN
	PackMLOut.eModePrevious	:= PackMLOut.eModeCurrent;
	PackMLOut.eModeCurrent	:= eNextMode;
	PackMLOut.bModeChanged	:= TRUE;
	H_OnModeChanged(PackMLOut.eModePrevious, PackMLOut.eModeCurrent);
END_IF
END_METHOD

METHOD PRIVATE M_ChangeState
VAR_INPUT
	eNextState	: E_PackMLState;
END_VAR
// Centralize state mutation so previous-state and edge outputs stay consistent.
IF PackMLOut.eStateCurrent <> eNextState THEN
	PackMLOut.eStatePrevious	:= PackMLOut.eStateCurrent;
	PackMLOut.eStateCurrent			:= eNextState;
	_bStateFirstScan			:= TRUE;
	H_OnStateChanged(PackMLOut.eStatePrevious, PackMLOut.eStateCurrent);
END_IF
END_METHOD

METHOD PRIVATE M_IsAbortAllowedByState : BOOL
// Abort is valid from every state except the terminal abort states.
M_IsAbortAllowedByState := (PackMLOut.eStateCurrent <> E_PackMLState.Aborting) AND (PackMLOut.eStateCurrent <> E_PackMLState.Aborted);
END_METHOD

METHOD PRIVATE M_IsClearAllowedByState : BOOL
// Clear leaves the safe Aborted state and starts the resettable stop path.
M_IsClearAllowedByState := PackMLOut.eStateCurrent = E_PackMLState.Aborted;
END_METHOD

METHOD PRIVATE M_IsCompleteAllowedByState : BOOL
// Complete is only meaningful while the unit is executing.
M_IsCompleteAllowedByState := PackMLOut.eStateCurrent = E_PackMLState.Execute;
END_METHOD

METHOD PRIVATE M_IsHoldAllowedByState : BOOL
// Hold pauses an active Execute flow.
M_IsHoldAllowedByState := PackMLOut.eStateCurrent = E_PackMLState.Execute;
END_METHOD

METHOD PRIVATE M_IsModeChangeAllowedByState : BOOL
// Mode changes can only be attempted from safe stable states.
// Target mode compatibility is checked separately after this safety gate.
// Henry: Bypass "Held" & "Suspended" state due to consideration about state-related parameters inconsistent
M_IsModeChangeAllowedByState :=
	(PackMLOut.eStateCurrent = E_PackMLState.Aborted) OR
	(PackMLOut.eStateCurrent = E_PackMLState.Stopped) OR
	(PackMLOut.eStateCurrent = E_PackMLState.Idle) OR
	(PackMLOut.eStateCurrent = E_PackMLState.Complete);
END_METHOD

METHOD PRIVATE M_IsResetAllowedByState : BOOL
// Reset prepares the unit from Stopped or Complete into Idle.
M_IsResetAllowedByState := (PackMLOut.eStateCurrent = E_PackMLState.Stopped) OR (PackMLOut.eStateCurrent = E_PackMLState.Complete);
END_METHOD

METHOD PRIVATE M_IsStartAllowedByState : BOOL
// Start begins production or operation only from Idle.
M_IsStartAllowedByState := PackMLOut.eStateCurrent = E_PackMLState.Idle;
END_METHOD

METHOD PRIVATE M_IsStopAllowedByState : BOOL
// Stop is accepted from normal operating, paused, and completing states.
M_IsStopAllowedByState :=
	(PackMLOut.eStateCurrent = E_PackMLState.Starting) OR
	(PackMLOut.eStateCurrent = E_PackMLState.Idle) OR
	(PackMLOut.eStateCurrent = E_PackMLState.Execute) OR
	(PackMLOut.eStateCurrent = E_PackMLState.Completing) OR
	(PackMLOut.eStateCurrent = E_PackMLState.Complete) OR
	(PackMLOut.eStateCurrent = E_PackMLState.Holding) OR
	(PackMLOut.eStateCurrent = E_PackMLState.Held) OR
	(PackMLOut.eStateCurrent = E_PackMLState.Unholding) OR
	(PackMLOut.eStateCurrent = E_PackMLState.Suspending) OR
	(PackMLOut.eStateCurrent = E_PackMLState.Suspended) OR
	(PackMLOut.eStateCurrent = E_PackMLState.Unsuspending);
END_METHOD

METHOD PRIVATE M_IsSuspendAllowedByState : BOOL
// Suspend pauses Execute because of an external process condition.
M_IsSuspendAllowedByState := PackMLOut.eStateCurrent = E_PackMLState.Execute;
END_METHOD

METHOD PRIVATE M_IsUnholdAllowedByState : BOOL
// Unhold resumes from the stable Held state.
M_IsUnholdAllowedByState := PackMLOut.eStateCurrent = E_PackMLState.Held;
END_METHOD

METHOD PRIVATE M_IsUnsuspendAllowedByState : BOOL
// Unsuspend resumes from the stable Suspended state.
M_IsUnsuspendAllowedByState := PackMLOut.eStateCurrent = E_PackMLState.Suspended;
END_METHOD

METHOD PRIVATE M_RejectCommand
VAR_INPUT
	eErrorID	: E_PackMLErrorID;
END_VAR
// Centralize rejected-command reporting so every guard failure has a stable ID.
PackMLOut.bCommandRejected	:= TRUE;
PackMLOut.eStateErrorID		:= eErrorID;
END_METHOD

METHOD PRIVATE M_RejectModeChange
VAR_INPUT
	eErrorID	: E_PackMLErrorID;
END_VAR
// Keep mode-change errors separate from PackML command/state errors.
PackMLOut.bModeChangeRejected	:= TRUE;
PackMLOut.eModeErrorID		:= eErrorID;
END_METHOD

// Used for requesting PackML command inside state machine itself 
METHOD PROTECTED FINAL RequestCommand : BOOL
VAR_INPUT
	eTargetCmd	: E_PackMLCommand;
END_VAR
RequestCommand := FALSE;

IF _bQueuedCommandRequest OR PackMLIn.bModeChangeRequest THEN
	RETURN;
END_IF

_eQueuedCommand			:= eTargetCmd;
_bQueuedCommandRequest	:= TRUE;
RequestCommand := TRUE;
END_METHOD

END_FUNCTION_BLOCK
